// TIA Portal V18 export
DATA_BLOCK "L1_gen"   // DB3
{ S7_Optimized_Access := 'TRUE' }
VERSION : 0.1
// stored: AutoNumber true, DBAccessibleFromOPCUA true, DBAccessibleFromWebserver true, IsOnlyStoredInLoadMemory false, IsRetainMemResEnabled false, IsWriteProtectedInAS false, MemoryReserve 100
   VAR RETAIN
      linea { S7_SetPoint := 'True'} : "LGasp_typeHMI_linea";
   END_VAR
BEGIN
   linea.NUMZONE := 5;
   linea.NUMDS := 50;
   linea.NUMSTAZIONI := 20;
   linea.NUMSAFETYDEVICE := 15;
   linea.NUMATTUATORI := 15;
   linea.NUMPUNZONATEARTICOLO := 100;
   linea.NUMRIGHEPRODUZIONE := 10;
   linea.NUMRIGHELISTATAGLI := 50;
   linea.NUMASSIAA := 3;
   linea.man := FALSE;
   linea.auto := FALSE;
   linea.semiauto := FALSE;
   linea.MARCIAstop := FALSE;
   linea.allarmi := TRUE;
   linea.warning := TRUE;
   linea.nome_linea := WSTRING#'210100008';
   linea.zona[1].abilitata := TRUE;
   linea.zona[2].abilitata := FALSE;
   linea.zona[3..4].abilitata := TRUE;
   linea.zona[5].abilitata := FALSE;
   linea.zona[1].nome := WSTRING#'Z1';
   linea.zona[2].nome := WSTRING#'Z2';
   linea.zona[3].nome := WSTRING#'Z3';
   linea.zona[4].nome := WSTRING#'Z4';
   linea.zona[5].nome := WSTRING#'Z5';
   linea.zona[1..5].AUTOman := FALSE;
   linea.zona[1..5].MARCIAstop := FALSE;
   linea.zona[1].allarmi := TRUE;
   linea.zona[2].allarmi := FALSE;
   linea.zona[3].allarmi := TRUE;
   linea.zona[4..5].allarmi := FALSE;
   linea.zona[1..5].warning := FALSE;
   linea.zona[1..5].fungointervenuto := FALSE;
   linea.zona[1..5].cancellointervenuto := FALSE;
   linea.zona[1].barrieraintervenuta := TRUE;
   linea.zona[2..5].barrieraintervenuta := FALSE;
   linea.zona[1].safetydevice[1..3].tipo := 1;
   linea.zona[1].safetydevice[4].tipo := 3;
   linea.zona[1].safetydevice[5].tipo := 5;
   linea.zona[1].safetydevice[6..15].tipo := 0;
   linea.zona[2].safetydevice[1..15].tipo := 0;
   linea.zona[3].safetydevice[1..3].tipo := 1;
   linea.zona[3].safetydevice[4..5].tipo := 5;
   linea.zona[3].safetydevice[6..9].tipo := 1;
   linea.zona[3].safetydevice[10..12].tipo := 5;
   linea.zona[3].safetydevice[13..15].tipo := 0;
   linea.zona[4].safetydevice[1..2].tipo := 1;
   linea.zona[4].safetydevice[3..5].tipo := 6;
   linea.zona[4].safetydevice[6..15].tipo := 0;
   linea.zona[5].safetydevice[1..15].tipo := 0;
   linea.zona[1].safetydevice[1].conn := WSTRING#'XC100';
   linea.zona[1].safetydevice[2].conn := WSTRING#'XC101';
   linea.zona[1].safetydevice[3].conn := WSTRING#'XC105';
   linea.zona[1].safetydevice[4].conn := WSTRING#'XC142';
   linea.zona[1].safetydevice[5].conn := WSTRING#'XC701';
   linea.zona[1].safetydevice[6..15].conn := WSTRING#'';
   linea.zona[2].safetydevice[1..15].conn := WSTRING#'';
   linea.zona[3].safetydevice[1].conn := WSTRING#'XC141';
   linea.zona[3].safetydevice[2].conn := WSTRING#'XC162';
   linea.zona[3].safetydevice[3].conn := WSTRING#'XC803';
   linea.zona[3].safetydevice[4].conn := WSTRING#'XC702';
   linea.zona[3].safetydevice[5].conn := WSTRING#'XC703';
   linea.zona[3].safetydevice[6].conn := WSTRING#'QE1';
   linea.zona[3].safetydevice[7].conn := WSTRING#'QE2';
   linea.zona[3].safetydevice[8].conn := WSTRING#'XC305';
   linea.zona[3].safetydevice[9].conn := WSTRING#'XC50';
   linea.zona[3].safetydevice[10].conn := WSTRING#'XC704';
   linea.zona[3].safetydevice[11].conn := WSTRING#'XC705';
   linea.zona[3].safetydevice[12].conn := WSTRING#'XC706';
   linea.zona[3].safetydevice[13..15].conn := WSTRING#'';
   linea.zona[4].safetydevice[1].conn := WSTRING#'XC400';
   linea.zona[4].safetydevice[2].conn := WSTRING#'XC406';
   linea.zona[4].safetydevice[3].conn := WSTRING#'XC707';
   linea.zona[4].safetydevice[4].conn := WSTRING#'XC708';
   linea.zona[4].safetydevice[5..15].conn := WSTRING#'';
   linea.zona[5].safetydevice[1..15].conn := WSTRING#'';
   linea.zona[1].safetydevice[1..3].intervenuto := FALSE;
   linea.zona[1].safetydevice[4].intervenuto := TRUE;
   linea.zona[1].safetydevice[5..15].intervenuto := FALSE;
   linea.zona[2].safetydevice[1].intervenuto := FALSE;
   linea.zona[2].safetydevice[2].intervenuto := TRUE;
   linea.zona[2].safetydevice[3..15].intervenuto := FALSE;
   linea.zona[3].safetydevice[1..15].intervenuto := FALSE;
   linea.zona[4].safetydevice[1..4].intervenuto := FALSE;
   linea.zona[4].safetydevice[5].intervenuto := TRUE;
   linea.zona[4].safetydevice[6..15].intervenuto := FALSE;
   linea.zona[5].safetydevice[1..2].intervenuto := FALSE;
   linea.zona[5].safetydevice[3..4].intervenuto := TRUE;
   linea.zona[5].safetydevice[5..15].intervenuto := FALSE;
   linea.zona[1].safetydevice[1..5].ninterventi := 2;
   linea.zona[1].safetydevice[6..15].ninterventi := 0;
   linea.zona[2].safetydevice[1].ninterventi := 4;
   linea.zona[2].safetydevice[2].ninterventi := 5;
   linea.zona[2].safetydevice[3].ninterventi := 4;
   linea.zona[2].safetydevice[4..7].ninterventi := 5;
   linea.zona[2].safetydevice[8..15].ninterventi := 0;
   linea.zona[3].safetydevice[1..8].ninterventi := 2;
   linea.zona[3].safetydevice[9].ninterventi := 3;
   linea.zona[3].safetydevice[10..12].ninterventi := 2;
   linea.zona[3].safetydevice[13..15].ninterventi := 0;
   linea.zona[4].safetydevice[1].ninterventi := 3;
   linea.zona[4].safetydevice[2..4].ninterventi := 2;
   linea.zona[4].safetydevice[5].ninterventi := 9;
   linea.zona[4].safetydevice[6..15].ninterventi := 0;
   linea.zona[5].safetydevice[1..2].ninterventi := 4;
   linea.zona[5].safetydevice[3].ninterventi := 7;
   linea.zona[5].safetydevice[4].ninterventi := 9;
   linea.zona[5].safetydevice[5..15].ninterventi := 0;
   linea.zona[1].safetydevice[1..15].dadefinire1 := 0;
   linea.zona[2].safetydevice[1..15].dadefinire1 := 0;
   linea.zona[3].safetydevice[1..15].dadefinire1 := 0;
   linea.zona[4].safetydevice[1..15].dadefinire1 := 0;
   linea.zona[5].safetydevice[1..15].dadefinire1 := 0;
   linea.zona[1].safetydevice[1..15].dadefinire2 := 0;
   linea.zona[2].safetydevice[1..15].dadefinire2 := 0;
   linea.zona[3].safetydevice[1..15].dadefinire2 := 0;
   linea.zona[4].safetydevice[1..15].dadefinire2 := 0;
   linea.zona[5].safetydevice[1..15].dadefinire2 := 0;
   linea.zona[1].safetydevice[1..15].dadefinire3 := 0;
   linea.zona[2].safetydevice[1..15].dadefinire3 := 0;
   linea.zona[3].safetydevice[1..15].dadefinire3 := 0;
   linea.zona[4].safetydevice[1..15].dadefinire3 := 0;
   linea.zona[5].safetydevice[1..15].dadefinire3 := 0;
   // linea.stz[1] : QUADRO
   // linea.stz[2] : PROFINET
   // linea.stz[3] : GENERALE
   // linea.stz[4] : ASPO+CULLA
   // linea.stz[5] : RADDRIZZATRICE
   // linea.stz[6] : GIUNZIONE
   // linea.stz[7] : ALIM+PUNZ
   // linea.stz[8] : PROFILA
   // linea.stz[9] : TAGLIO
   // linea.stz[10] : SCARICO
   linea.stz[1..10].abilitata := TRUE;
   linea.stz[11..20].abilitata := FALSE;
   linea.stz[1..2].invisibile := TRUE;
   linea.stz[3..5].invisibile := FALSE;
   linea.stz[6..7].invisibile := TRUE;
   linea.stz[8..9].invisibile := FALSE;
   linea.stz[10..20].invisibile := TRUE;
   linea.stz[1..3].zona := 3;
   linea.stz[4].zona := 1;
   linea.stz[5..7].zona := 2;
   linea.stz[8].zona := 3;
   linea.stz[9].zona := 4;
   linea.stz[10..20].zona := 5;
   linea.stz[1].nome := WSTRING#'STZ QUADRO';
   linea.stz[2].nome := WSTRING#'STZ PROFINET';
   linea.stz[3].nome := WSTRING#'STZ GENERALE';
   linea.stz[4].nome := WSTRING#'STZ ASPO+CULLA';
   linea.stz[5].nome := WSTRING#'STZ RADDRIZZATRICE';
   linea.stz[6].nome := WSTRING#'STZ GIUNZIONE';
   linea.stz[7].nome := WSTRING#'STZ ALIM+PUNZ';
   linea.stz[8].nome := WSTRING#'STZ PROFILA';
   linea.stz[9].nome := WSTRING#'STZ TAGLIO';
   linea.stz[10].nome := WSTRING#'STZ SCARICO';
   linea.stz[11..20].nome := WSTRING#'';
   linea.stz[1].nometrad := WSTRING#'QUADRO';
   linea.stz[2].nometrad := WSTRING#'PROFINET';
   linea.stz[3].nometrad := WSTRING#'GENERALE';
   linea.stz[4].nometrad := WSTRING#'ASPO';
   linea.stz[5].nometrad := WSTRING#'RADDRIZZATRICE';
   linea.stz[6].nometrad := WSTRING#'GIUNZIONE';
   linea.stz[7].nometrad := WSTRING#'ALIM + PUNZ';
   linea.stz[8].nometrad := WSTRING#'PROFILA';
   linea.stz[9].nometrad := WSTRING#'TAGLIO';
   linea.stz[10].nometrad := WSTRING#'SCARICO';
   linea.stz[11].nometrad := WSTRING#'AGGRAFFATURA';
   linea.stz[12..19].nometrad := WSTRING#'DISPONIBILE';
   linea.stz[20].nometrad := WSTRING#'';
   linea.stz[1..20].AUTOman := FALSE;
   linea.stz[1..20].MARCIAstop := FALSE;
   linea.stz[1..2].allarmi := FALSE;
   linea.stz[3..4].allarmi := TRUE;
   linea.stz[5..7].allarmi := FALSE;
   linea.stz[8].allarmi := TRUE;
   linea.stz[9..20].allarmi := FALSE;
   linea.stz[1..3].warning := FALSE;
   linea.stz[4].warning := TRUE;
   linea.stz[5..20].warning := FALSE;
   // linea.stz[4].ds[1] : L1-ASPO- DIAMETRO COIL-DISTANZA LASER CENTRO ASPO [mm]
   // linea.stz[4].ds[2] : L1-ASPO- ANSA XC142A-1-SOGLIA BASSA [mm]
   // linea.stz[4].ds[3] : L1-ASPO- ANSA XC142A-1-SOGLIA ALTA [mm]
   // linea.stz[4].ds[5] : L1-ASPO-FRENATURA-COPPIA MAX [%]
   // linea.stz[4].ds[6] : L1-ASPO-FRENATURA-VELOCITA' AUTOMATICA [%]
   // linea.stz[4].ds[8] : L1-ASPO-M101 MADRINO -VELOCITA' MANUALE [%]
   // linea.stz[4].ds[15] : L1-ASPO-M101 MADRINO -INTERVALLO PER ESPANSIONE AUTOMATICA [min]
   // linea.stz[4].ds[16] : L1-ASPO-M101 MADRINO -DURATA ESPANSIONE AUTOMATICA [sec]
   // linea.stz[5].ds[1] : L1-RADDRIZZATRICE-ANSA-VELOCITA' BASSA [%]
   // linea.stz[5].ds[2] : L1-RADDRIZZATRICE-ANSA-VELOCITA' MEDIA [%]
   // linea.stz[5].ds[3] : L1-RADDRIZZATRICE-ANSA-VELOCITA' ALTA [%]
   // linea.stz[5].ds[4] : L1-RADDRIZZATRICE-ANSA-SOGLIA BASSA [mm]
   // linea.stz[5].ds[5] : L1-RADDRIZZATRICE-ANSA-SOGLIA INTEMEDIA BASSA [mm]
   // linea.stz[5].ds[6] : L1-RADDRIZZATRICE-ANSA-SOGLIA INTEMEDIA ALTA [mm]
   // linea.stz[5].ds[7] : L1-RADDRIZZATRICE-ANSA-SOGLIA ALTA [mm]
   // linea.stz[5].ds[8] : L1-RADDRIZZATRICE-M141-VELOCITA' MANUALE [%]
   // linea.stz[7].ds[1] : L1-ALIM + PUNZ-M201-ALIMENTATORE A RULLI-VELOCITA' MANUALE [%]
   // linea.stz[7].ds[2] : L1-ALIM + PUNZ-M201-ALIMENTATORE A RULLI-VELOCITA QUOTA FINE PRODUZIONE [%]
   // linea.stz[7].ds[3] : L1-ALIM + PUNZ-M201-ALIMENTATORE A RULLI-DISTANZA LAMA-GIUNZIONE CON PUNTO DI SALDATURA [mm]
   // linea.stz[7].ds[4] : L1-ALIM + PUNZ-M201-ALIMENTATORE A RULLI-QUOTA ALIMENTATORE A FINE PRODUZIONE [mm]
   // linea.stz[7].ds[5] : L1-ALIM + PUNZ-ANSA-SOGLIA BASSA [mm]
   // linea.stz[7].ds[6] : L1-ALIM + PUNZ-ANSA-SOGLIA INTEMEDIA BASSA [mm]
   // linea.stz[7].ds[7] : L1-ALIM + PUNZ-ANSA-SOGLIA INTEMEDIA ALTA [mm]
   // linea.stz[7].ds[8] : L1-ALIM + PUNZ-ANSA-SOGLIA ALTA [mm]
   // linea.stz[7].ds[9] : L1-ALIM + PUNZ-PRESSA-VELOCITA MANUALE-SEMIAUTO [%]
   // linea.stz[7].ds[10] : L1-ALIM + PUNZ-PRESSA-OFFSET ENCODER ASSOLUTO
   // linea.stz[7].ds[11] : L1-ALIM + PUNZ-PRESSA-ANGOLO INIZIO PMS [°]
   // linea.stz[7].ds[12] : L1-ALIM + PUNZ-PRESSA-ANGOLO FINE PMS [°]
   // linea.stz[7].ds[13] : L1-ALIM + PUNZ-PRESSA-ANGOLO INIZIO PMI [°]
   // linea.stz[7].ds[14] : L1-ALIM + PUNZ-PRESSA-ANGOLO FINE PMI [°]
   // linea.stz[7].ds[15] : L1-ALIM + PUNZ-PRESSA-ANGOLO INIZIO AREA DI LAVORO [°]
   // linea.stz[7].ds[16] : L1-ALIM + PUNZ-PRESSA-ANGOLO FINE AREA DI LAVORO [°]
   // linea.stz[7].ds[17] : L1-ALIM + PUNZ-PRESSA-NUMERO COLPI IN SEMI AUTOMATICO
   // linea.stz[7].ds[18] : L1-ALIM + PUNZ-DROPSA-NUMERO COLPI PER LUBRIFICAZIONE
   // linea.stz[7].ds[19] : L1-ALIM + PUNZ-DROPSA-DURATA LUBRIFICAZIONE [sec]
   // linea.stz[8].ds[1] : L1-PROFILA-M301 PROFILA-VELOCITA' MANUALE [%]
   // linea.stz[8].ds[2] : L1-PROFILA-M301 PROFILA-VELOCITA SVUOTAMENTO [%]
   // linea.stz[8].ds[4] : L1-PROFILA-M365 ESTRATTORE-VELOCITA' MANUALE [%]
   // linea.stz[8].ds[8] : L1-PROFILA-SALDATRICE-POTENZA SALDATURA [%]
   // linea.stz[8].ds[11] : L1-PROFILA-QUOTA ATTIVAZIONE LUBRIFICAZIONE [mm]
   // linea.stz[8].ds[12] : L1-PROFILA-DURATA LUBRIFICAZIONE [sec]
   // linea.stz[9].ds[2] : L1-TAGLIO-DURATA LUBRIFICAZIONE [sec]
   // linea.stz[9].ds[3] : L1-TAGLIO-NUMERO COLPI PER LUBRIFICAZIONE
   // linea.stz[9].ds[4] : L1-TAGLIO-M404 SALITA DISCESA DISCO TAGLIO-VELOCITA' MANUALE [%]
   // linea.stz[9].ds[6] : L1-TAGLIO-M405 ROTAZIONE DISCO TAGLIO-VELOCITA' MANUALE [%]
   // linea.stz[9].ds[7] : L1-TAGLIO-M405 ROTAZIONE DISCO TAGLIO-VELOCITA' SPESSORE 0.5-0.6
   // linea.stz[9].ds[8] : L1-TAGLIO-M405 ROTAZIONE DISCO TAGLIO-VELOCITA' SPESSORE 0.8-1.0
   // linea.stz[9].ds[9] : L1-TAGLIO-M405 ROTAZIONE DISCO TAGLIO-VELOCITA' SPESSORE 1.2-1.5
   // linea.stz[9].ds[10] : L1-TAGLIO-M404 SALITA DISCESA DISCO TAGLIO-POSIZIONE PUNTO MORTO SUP [mm]
   // linea.stz[9].ds[11] : L1-TAGLIO-M404 SALITA DISCESA DISCO TAGLIO-POSIZIONE PUNTO MORTO INF [mm]
   // linea.stz[9].ds[12] : L1-TAGLIO-M404 SALITA DISCESA DISCO TAGLIO-POSIZIONE CAMBIO LAMA [mm]
   // linea.stz[9].ds[13] : L1-TAGLIO-M404 SALITA DISCESA DISCO TAGLIO-VELOCITA' SPESSORE 0.5-0.6
   // linea.stz[9].ds[14] : L1-TAGLIO-M404 SALITA DISCESA DISCO TAGLIO-VELOCITA' SPESSORE 0.8-1.0
   // linea.stz[9].ds[15] : L1-TAGLIO-M404 SALITA DISCESA DISCO TAGLIO-VELOCITA' SPESSORE 1.2-1.5
   // linea.stz[9].ds[16] : L1-TAGLIO-M404 SALITA DISCESA DISCO TAGLIO-VELOCITA' SALITA
   // linea.stz[9].ds[17] : L1-TAGLIO-M401 CARRO TAGLIO AL VOLO-DISTANZA LASER LAMA DI TAGLIO[mm]
   // linea.stz[9].ds[19] : L1-TAGLIO-M408 TAPPETO EVACUAZIONE-VELOCITA INTERMEDIA [%]
   // linea.stz[9].ds[20] : L1-TAGLIO-M408 TAPPETO EVACUAZIONE-VELOCITA' ALTA [%]
   // linea.stz[9].ds[21] : L1-TAGLIO-M408 TAPPETO EVACUAZIONE-VELOCITA' MANUALE [%]
   linea.stz[1].ds[1..50].val := 0.0;
   linea.stz[2].ds[1..50].val := 0.0;
   linea.stz[3].ds[1..50].val := 0.0;
   linea.stz[4].ds[1].val := 2090.0;
   linea.stz[4].ds[2..4].val := 0.0;
   linea.stz[4].ds[5].val := 10.0;
   linea.stz[4].ds[6].val := 1.0;
   linea.stz[4].ds[7].val := 0.0;
   linea.stz[4].ds[8..9].val := 10.0;
   linea.stz[4].ds[10..12].val := 25.0;
   linea.stz[4].ds[13..14].val := 0.0;
   linea.stz[4].ds[15].val := 5.0;
   linea.stz[4].ds[16].val := 60.0;
   linea.stz[4].ds[17].val := 0.0;
   linea.stz[4].ds[18].val := 5.0;
   linea.stz[4].ds[19].val := 60.0;
   linea.stz[4].ds[20..50].val := 0.0;
   linea.stz[5].ds[1].val := 5.0;
   linea.stz[5].ds[2].val := 50.0;
   linea.stz[5].ds[3].val := 80.0;
   linea.stz[5].ds[4].val := 2300.0;
   linea.stz[5].ds[5].val := 2200.0;
   linea.stz[5].ds[6].val := 2000.0;
   linea.stz[5].ds[7].val := 1700.0;
   linea.stz[5].ds[8].val := 80.0;
   linea.stz[5].ds[9..50].val := 0.0;
   linea.stz[6].ds[1..50].val := 0.0;
   linea.stz[7].ds[1].val := 20.0;
   linea.stz[7].ds[2..4].val := 0.0;
   linea.stz[7].ds[5].val := 2300.0;
   linea.stz[7].ds[6].val := 2200.0;
   linea.stz[7].ds[7].val := 2000.0;
   linea.stz[7].ds[8].val := 1700.0;
   linea.stz[7].ds[9].val := 60.0;
   linea.stz[7].ds[10].val := -214.0;
   linea.stz[7].ds[11].val := 340.0;
   linea.stz[7].ds[12].val := 20.0;
   linea.stz[7].ds[13].val := 160.0;
   linea.stz[7].ds[14].val := 200.0;
   linea.stz[7].ds[15].val := 130.0;
   linea.stz[7].ds[16].val := 230.0;
   linea.stz[7].ds[17].val := 60.0;
   linea.stz[7].ds[18..50].val := 0.0;
   linea.stz[8].ds[1].val := 15.0;
   linea.stz[8].ds[2].val := 10.0;
   linea.stz[8].ds[3..4].val := 0.0;
   linea.stz[8].ds[5].val := 10000.0;
   linea.stz[8].ds[6].val := 30.0;
   linea.stz[8].ds[7].val := 0.0;
   linea.stz[8].ds[8].val := 90.0;
   linea.stz[8].ds[9..10].val := 0.0;
   linea.stz[8].ds[11].val := 60.0;
   linea.stz[8].ds[12..13].val := 1.0;
   linea.stz[8].ds[14..50].val := 0.0;
   linea.stz[9].ds[1..50].val := 0.0;
   linea.stz[10].ds[1..50].val := 0.0;
   linea.stz[11].ds[1..50].val := 0.0;
   linea.stz[12].ds[1..50].val := 0.0;
   linea.stz[13].ds[1..50].val := 0.0;
   linea.stz[14].ds[1..50].val := 0.0;
   linea.stz[15].ds[1..50].val := 0.0;
   linea.stz[16].ds[1..50].val := 0.0;
   linea.stz[17].ds[1..50].val := 0.0;
   linea.stz[18].ds[1..50].val := 0.0;
   linea.stz[19].ds[1..50].val := 0.0;
   linea.stz[20].ds[1..50].val := 0.0;
   linea.stz[1].ds[1..50].ll := 0.0;
   linea.stz[2].ds[1..50].ll := 0.0;
   linea.stz[3].ds[1..50].ll := 0.0;
   linea.stz[4].ds[1..4].ll := 0.0;
   linea.stz[4].ds[5..6].ll := 1.0;
   linea.stz[4].ds[7..9].ll := 0.0;
   linea.stz[4].ds[10..12].ll := 1.0;
   linea.stz[4].ds[13..50].ll := 0.0;
   linea.stz[5].ds[1..50].ll := 0.0;
   linea.stz[6].ds[1..50].ll := 0.0;
   linea.stz[7].ds[1..9].ll := 0.0;
   linea.stz[7].ds[10].ll := -360.0;
   linea.stz[7].ds[11..16].ll := 0.0;
   linea.stz[7].ds[17].ll := 40.0;
   linea.stz[7].ds[18..50].ll := 0.0;
   linea.stz[8].ds[1..2].ll := 1.0;
   linea.stz[8].ds[3..5].ll := 0.0;
   linea.stz[8].ds[6].ll := 1.0;
   linea.stz[8].ds[7].ll := 0.0;
   linea.stz[8].ds[8].ll := 1.0;
   linea.stz[8].ds[9..12].ll := 0.0;
   linea.stz[8].ds[13].ll := 0.9;
   linea.stz[8].ds[14..50].ll := 0.0;
   linea.stz[9].ds[1..50].ll := 0.0;
   linea.stz[10].ds[1..50].ll := 0.0;
   linea.stz[11].ds[1..50].ll := 0.0;
   linea.stz[12].ds[1..50].ll := 0.0;
   linea.stz[13].ds[1..50].ll := 0.0;
   linea.stz[14].ds[1..50].ll := 0.0;
   linea.stz[15].ds[1..50].ll := 0.0;
   linea.stz[16].ds[1..50].ll := 0.0;
   linea.stz[17].ds[1..50].ll := 0.0;
   linea.stz[18].ds[1..50].ll := 0.0;
   linea.stz[19].ds[1..50].ll := 0.0;
   linea.stz[20].ds[1..50].ll := 0.0;
   linea.stz[1].ds[1..50].hl := 0.0;
   linea.stz[2].ds[1..50].hl := 0.0;
   linea.stz[3].ds[1..50].hl := 0.0;
   linea.stz[4].ds[1].hl := 3000.0;
   linea.stz[4].ds[2..4].hl := 0.0;
   linea.stz[4].ds[5..6].hl := 100.0;
   linea.stz[4].ds[7].hl := 0.0;
   linea.stz[4].ds[8..12].hl := 100.0;
   linea.stz[4].ds[13..14].hl := 0.0;
   linea.stz[4].ds[15].hl := 60.0;
   linea.stz[4].ds[16].hl := 200.0;
   linea.stz[4].ds[17].hl := 0.0;
   linea.stz[4].ds[18].hl := 60.0;
   linea.stz[4].ds[19].hl := 200.0;
   linea.stz[4].ds[20..50].hl := 0.0;
   linea.stz[5].ds[1..3].hl := 100.0;
   linea.stz[5].ds[4..7].hl := 2400.0;
   linea.stz[5].ds[8].hl := 100.0;
   linea.stz[5].ds[9..50].hl := 0.0;
   linea.stz[6].ds[1..50].hl := 0.0;
   linea.stz[7].ds[1].hl := 100.0;
   linea.stz[7].ds[2..4].hl := 0.0;
   linea.stz[7].ds[5..8].hl := 2400.0;
   linea.stz[7].ds[9].hl := 100.0;
   linea.stz[7].ds[10..16].hl := 360.0;
   linea.stz[7].ds[17].hl := 100.0;
   linea.stz[7].ds[18..50].hl := 0.0;
   linea.stz[8].ds[1..2].hl := 100.0;
   linea.stz[8].ds[3..4].hl := 0.0;
   linea.stz[8].ds[5].hl := 20000.0;
   linea.stz[8].ds[6].hl := 100.0;
   linea.stz[8].ds[7].hl := 0.0;
   linea.stz[8].ds[8].hl := 100.0;
   linea.stz[8].ds[9..10].hl := 0.0;
   linea.stz[8].ds[11].hl := 120.0;
   linea.stz[8].ds[12].hl := 60.0;
   linea.stz[8].ds[13].hl := 1.1;
   linea.stz[8].ds[14..50].hl := 0.0;
   linea.stz[9].ds[1..22].hl := 0.0;
   linea.stz[9].ds[23].hl := 2000.0;
   linea.stz[9].ds[24..50].hl := 0.0;
   linea.stz[10].ds[1..50].hl := 0.0;
   linea.stz[11].ds[1..50].hl := 0.0;
   linea.stz[12].ds[1..50].hl := 0.0;
   linea.stz[13].ds[1..50].hl := 0.0;
   linea.stz[14].ds[1..50].hl := 0.0;
   linea.stz[15].ds[1..50].hl := 0.0;
   linea.stz[16].ds[1..50].hl := 0.0;
   linea.stz[17].ds[1..50].hl := 0.0;
   linea.stz[18].ds[1..50].hl := 0.0;
   linea.stz[19].ds[1..50].hl := 0.0;
   linea.stz[20].ds[1..50].hl := 0.0;
   linea.stz[1].all[1] := FALSE;   // L1-QUADRO[1]- 24-L4+ EMERGENZA GENERALE
   linea.stz[1].all[2] := FALSE;   // L1-QUADRO[2]-
   linea.stz[1].all[3] := FALSE;   // L1-QUADRO[3]-D6-QF1-PROTEZIONE INTERVENUTA PRIMARIO TRASFORMATORE 400:230V
   linea.stz[1].all[4] := FALSE;   // L1-QUADRO[4]-D6-QF2-PROTEZIONE INTERVENUTA SECONDARIO TRASFORMATORE 400:230V
   linea.stz[1].all[5] := FALSE;
   linea.stz[1].all[6] := FALSE;   // L1-QUADRO[6]-D8-FU1 24-L1+-PROTEZIONE ELETTRONICA INTERVENUTA ALIMENTAZIONE Q.E.
   linea.stz[1].all[7] := FALSE;   // L1-QUADRO[7]-D8 FU1 24-L3+-PROTEZIONE ELETTRONICA INTERVENUTA ALIMENTAZIONE PULSANTIERE
   linea.stz[1].all[8] := FALSE;   // L1-QUADRO[8]-D8 FU1 24-L3+S-PROTEZIONE ELETTRONICA INTERVENUTA ALIMENTAZIONE SICUREZZE
   linea.stz[1].all[9] := FALSE;   // L1-QUADRO[9]-D8 FU1 24-L3+1-PROTEZIONE ELETTRONICA INTERVENUTA ALIMENTAZIONE B.M.1 (MANDRINI ASPO)
   linea.stz[1].all[10] := FALSE;   // L1-QUADRO[10]-D8 FU1 24-L3+2-PROTEZIONE ELETTRONICA INTERVENUTA ALIMENTAZIONE B.M. 2 (TIN + RADDRIZZATRICE- + CENTRALE PROFILA)
   linea.stz[1].all[11] := FALSE;   // L1-QUADRO[11]-D8 FU1 24-L3+3-PROTEZIONE ELETTRONICA INTERVENUTA ALIMENTAZIONE B.M. 3 (VASCA LIQUIDO)
   linea.stz[1].all[12] := FALSE;   // L1-QUADRO[12]-D8 FU1 24-L10+-PROTEZIONE ELETTRONICA INTERVENUTA ALIMENTAZIONE PC
   linea.stz[1].all[13] := FALSE;   // L1-QUADRO[13]-D8 FU1 24-L11+ PROTEZIONE ELETTRONICA INTERVENUTA ALIMENTAZIONE NODI IN Q.E.
   linea.stz[1].all[14] := FALSE;   // L1-QUADRO[14]-D9 FU1 24-L13+ -PROTEZIONE ELETTRONICA INTERVENUTA ALIMENTAZIONE LOGICA AZIONAMENTI
   linea.stz[1].all[15] := FALSE;   // L1-QUADRO[15]-D9 FU1 24-L131+ -PROTEZIONE ELETTRONICA INTERVENUTA ALIMENTAZIONE LOGICA ALIMENTATORE 45KW
   linea.stz[1].all[16] := FALSE;   // L1-QUADRO[16]-D9 FU124-L3+4 PROTEZIONE ELETTRONICA INTERVENUTA ALIMENTAZIONE B.M. 4 (TAGLIO + CENTRALE IDRAULICA)
   linea.stz[1].all[17] := FALSE;   // L1-QUADRO[17]-D17 FU1 OUT 4 (PREDISPOSTO)
   linea.stz[1].all[18] := FALSE;   // L1-QUADRO[18]-D16 FU1 24-L4+ PROTEZIONE ELETTRONICA INTERVENUTA - EMERGENZA GENERALE
   linea.stz[1].all[19] := FALSE;   // L1-QUADRO[19]-D16 FU1 24-L41+ PROTEZIONE ELETTRONICA INTERVENUTA - EMERGENZA ISTANTANEA ZONA 1 (SVOLGITURA)
   linea.stz[1].all[20] := FALSE;   // L1-QUADRO[20]-D16 FU1 24-L42+ PROTEZIONE ELETTRONICA INTERVENUTA - EMERGENZA ISTANTANEA ZONA 2 (GIUNZIONE)
   linea.stz[1].all[21] := FALSE;   // L1-QUADRO[21]-D16 FU1 24-L44+ PROTEZIONE ELETTRONICA INTERVENUTA - EMERGENZA ISTANTANEA ZONA 4 TAGLIO)
   linea.stz[1].all[22] := FALSE;   // L1-QUADRO[22]-D16 FU1 24-L43+ PROTEZIONE ELETTRONICA INTERVENUTA - EMERGENZA ISTANTANEA ZONA 3 PROFILA)
   linea.stz[1].all[23] := FALSE;   // L1-QUADRO[23]-D16 FU1 24-L411+ PROTEZIONE ELETTRONICA INTERVENUTA - EMERGENZA ISTANTANEA ZONA 1 MANDRINO 1)
   linea.stz[1].all[24] := FALSE;   // L1-QUADRO[24]-D16 FU1 24-L412+ PROTEZIONE ELETTRONICA INTERVENUTA - EMERGENZA ISTANTANEA ZONA 1 MANDRINO 2)
   linea.stz[1].all[25] := FALSE;   // L1-QUADRO[25]-D16 FU1 24-L4+3 PROTEZIONE ELETTRONICA INTERVENUTA - EMERGENZA ISTANTANEA
   linea.stz[1].all[26] := FALSE;   // L1-QUADRO[26]-D17 FU1 24-L4+1 PROTEZIONE ELETTRONICA INTERVENUTA - EMERGENZA ISTANTANEA
   linea.stz[1].all[27] := FALSE;   // L1-QUADRO[27]-D17 FU1 24-L4+2 PROTEZIONE ELETTRONICA INTERVENUTA - EMERGENZA ISTANTANEA
   linea.stz[1].all[28] := FALSE;   // L1-QUADRO[28]-D17 FU1 24-L43+1 PROTEZIONE ELETTRONICA INTERVENUTA - EMERGENZA ISTANTANEA
   linea.stz[1].all[29] := FALSE;   // L1-QUADRO[29]-D17 OUT 4 PREDISPOSTO
   linea.stz[1].all[30] := FALSE;   // L1-QUADRO[30]-D7-QF1 TERMICA ALIMENTATORE LINEA 24VDC INGRESSI
   linea.stz[1].all[31] := FALSE;   // L1-QUADRO[31]- D15-QF1 TERMICA ALIMENTATORE LINEA 24VDC USCITE
   linea.stz[1].all[32] := FALSE;   // L1-QUADRO[32]-D21-QF1 LINEA TERMICA PRESE QUADRO ELETTRICO
   linea.stz[1].all[33] := FALSE;   // L1-QUADRO[33]- D23-QF1 TERMICA VENTILAZIONE QUADRO
   linea.stz[1].all[34] := FALSE;   // L1-QUADRO[34]- D15-UV1 ANOMALIA ALIMENTATORE 1
   linea.stz[1].all[35] := FALSE;   // L1-QUADRO[35]- D15-UV2 ANOMALIA ALIMENTATORE 2
   linea.stz[1].all[36] := FALSE;   // L1-QUADRO[36]-
   linea.stz[1].all[37] := FALSE;   // L1-QUADRO[37]-
   linea.stz[1].all[38] := FALSE;   // L1-QUADRO[38]- G13-QF361 TERMICA MOTORE POMPA MANDATA LUBROREFRIGERAZIONE
   linea.stz[1].all[39] := FALSE;   // L1-QUADRO[39]- G14-QF368 TERMICA MOTORE POMPA SOMMERSA LUBROREFRIGERAZIONE
   linea.stz[1].all[40] := FALSE;   // L1-QUADRO[40]-
   linea.stz[1].all[41] := FALSE;   // L1-QUADRO[41]-
   linea.stz[1].all[42] := FALSE;   // L1-QUADRO[42]-
   linea.stz[1].all[43] := FALSE;   // L1-QUADRO[43]-
   linea.stz[1].all[44] := FALSE;   // L1-QUADRO[44]- M7-BT1- ALTA TEMPERATURA
   linea.stz[1].all[45] := FALSE;   // L1-QUADRO[45]-
   linea.stz[1].all[46] := FALSE;   // L1-QUADRO[46]-
   linea.stz[1].all[47] := FALSE;   // L1-QUADRO[47]-
   linea.stz[1].all[48] := FALSE;   // L1-QUADRO[48]-
   linea.stz[1].all[49] := FALSE;   // L1-QUADRO[49]-
   linea.stz[1].all[50] := FALSE;   // L1-QUADRO[50]-
   linea.stz[1].all[51] := FALSE;   // L1-QUADRO[51]-
   linea.stz[1].all[52] := FALSE;   // L1-QUADRO[52]
   linea.stz[1].all[53] := FALSE;   // L1-QUADRO[53]
   linea.stz[1].all[54] := FALSE;   // L1-QUADRO[54]-
   linea.stz[1].all[55..59] := FALSE;
   linea.stz[1].all[60] := FALSE;   // L1-QUADRO[60]-M9-M112-141DRV SOGLIA CARICO TERMICO RESISTENZA FRENATURA TORRETTA E RADDRIZZATORE
   linea.stz[1].all[61] := FALSE;   // L1-QUADRO[61]-M9-M102DRV SOGLIA CARICO TERMICO RESISTENZA FRENATURA ROTAZIONE MANDRINO 2
   linea.stz[1].all[62] := FALSE;   // L1-QUADRO[62]-M9-M101DRV SOGLIA CARICO TERMICO RESISTENZA FRENATURA ROTAZIONE MANDRINO 1
   linea.stz[1].all[63] := FALSE;   // L1-QUADRO[63]-M9-M401DRV SOGLIA CARICO TERMICO RESISTENZA FRENATURA TAGLIO ALVOLO
   linea.stz[1].all[64] := FALSE;   // L1-QUADRO[64]-M9-K30A1 ALTA TEMPERATURA ALIMENTATORE DRIVER 120KW
   linea.stz[1].all[65] := FALSE;   // L1-QUADRO[65]-M9-K30A1 ALIMENTATORE DRIVER BUS DC 120KW NON OK
   linea.stz[1].all[66] := FALSE;   // L1-QUADRO[66]-M9-K30A1 ALIMENTATORE DRIVER 120KW NON OK
   linea.stz[1].all[67] := FALSE;   // L1-QUADRO[67]-M10-M301DRV SOGLIA CARICO TERMICO RESISTENZA FRENATURA PROFILA MOTORE 1
   linea.stz[1].all[68] := FALSE;   // L1-QUADRO[68]-M10-M302DRV SOGLIA CARICO TERMICO RESISTENZA FRENATURA PROFILA MOTORE 2
   linea.stz[1].all[69] := FALSE;   // L1-QUADRO[69]-M10-M303DRV SOGLIA CARICO TERMICO RESISTENZA FRENATURA PROFILA MOTORE 3
   linea.stz[1].all[70] := FALSE;   // L1-QUADRO[70]- DIFFERENZIALE INTERVENUTO
   linea.stz[1].all[71] := FALSE;   // L1-QUADRO[71]-
   linea.stz[1].all[72] := FALSE;   // L1-QUADRO[72]-
   linea.stz[1].all[73] := FALSE;   // L1-QUADRO[73]-
   linea.stz[1].all[74] := FALSE;   // L1-QUADRO[74]-
   linea.stz[1].all[75] := FALSE;   // L1-QUADRO[75]-
   linea.stz[1].all[76] := FALSE;   // L1-QUADRO[76]-
   linea.stz[1].all[77] := FALSE;   // L1-QUADRO[77]-
   linea.stz[1].all[78] := FALSE;   // L1-QUADRO[78]-
   linea.stz[1].all[79] := FALSE;   // L1-QUADRO[79]-
   linea.stz[1].all[80] := FALSE;   // L1-QUADRO[80]-
   linea.stz[1].all[81..192] := FALSE;
   linea.stz[2].all[1] := FALSE;   // L1-PROFINET[1]
   linea.stz[2].all[2] := FALSE;   // L1-PROFINET[2]
   linea.stz[2].all[3] := FALSE;   // L1-PROFINET[3]
   linea.stz[2].all[4] := FALSE;   // L1-PROFINET[4]
   linea.stz[2].all[5] := FALSE;   // L1-PROFINET[5]
   linea.stz[2].all[6] := FALSE;   // L1-PROFINET[6]
   linea.stz[2].all[7] := FALSE;   // L1-PROFINET[7]
   linea.stz[2].all[8] := FALSE;   // L1-PROFINET[8]
   linea.stz[2].all[9] := FALSE;   // L1-PROFINET[9]
   linea.stz[2].all[10] := FALSE;   // L1-PROFINET[10]
   linea.stz[2].all[11] := FALSE;   // L1-PROFINET[11]
   linea.stz[2].all[12] := FALSE;   // L1-PROFINET[12]-ERRORE COMUNICAZIONE
   linea.stz[2].all[13] := FALSE;   // L1-PROFINET[13]
   linea.stz[2].all[14] := FALSE;   // L1-PROFINET[14]
   linea.stz[2].all[15] := FALSE;   // L1-PROFINET[15]
   linea.stz[2].all[16] := FALSE;   // L1-PROFINET[16]
   linea.stz[2].all[17] := FALSE;   // L1-PROFINET[17]
   linea.stz[2].all[18] := FALSE;   // L1-PROFINET[18]
   linea.stz[2].all[19] := FALSE;   // L1-PROFINET[19]
   linea.stz[2].all[20] := FALSE;   // L1-PROFINET[20]-ERRORE COMUNICAZIONE
   linea.stz[2].all[21] := FALSE;   // L1-PROFINET[21]-ERRORE COMUNICAZIONE
   linea.stz[2].all[22] := FALSE;   // L1-PROFINET[22]-ERRORE COMUNICAZIONE
   linea.stz[2].all[23] := FALSE;   // L1-PROFINET[23]-ERRORE COMUNICAZIONE
   linea.stz[2].all[24] := FALSE;   // L1-PROFINET[24]-ERRORE COMUNICAZIONE
   linea.stz[2].all[25] := FALSE;   // L1-PROFINET[25]
   linea.stz[2].all[26] := FALSE;   // L1-PROFINET[26]-ERRORE COMUNICAZIONE
   linea.stz[2].all[27] := FALSE;   // L1-PROFINET[27]
   linea.stz[2].all[28] := FALSE;   // L1-PROFINET[28]
   linea.stz[2].all[29] := FALSE;   // L1-PROFINET[29]
   linea.stz[2].all[30] := FALSE;   // L1-PROFINET[30]
   linea.stz[2].all[31] := FALSE;   // L1-PROFINET[31]
   linea.stz[2].all[32] := FALSE;   // L1-PROFINET[32]
   linea.stz[2].all[33] := FALSE;   // L1-PROFINET[33]
   linea.stz[2].all[34] := FALSE;   // L1-PROFINET[34]
   linea.stz[2].all[35] := FALSE;   // L1-PROFINET[35]
   linea.stz[2].all[36] := FALSE;   // L1-PROFINET[36]
   linea.stz[2].all[37] := FALSE;   // L1-PROFINET[37]
   linea.stz[2].all[38] := FALSE;   // L1-PROFINET[38]
   linea.stz[2].all[39] := FALSE;   // L1-PROFINET[39]
   linea.stz[2].all[40] := FALSE;   // L1-PROFINET[40]
   linea.stz[2].all[41] := FALSE;   // L1-PROFINET[41]
   linea.stz[2].all[42] := FALSE;   // L1-PROFINET[42]
   linea.stz[2].all[43] := FALSE;   // L1-PROFINET[43]
   linea.stz[2].all[44] := FALSE;   // L1-PROFINET[44]
   linea.stz[2].all[45] := FALSE;   // L1-PROFINET[45]
   linea.stz[2].all[46] := FALSE;   // L1-PROFINET[46]
   linea.stz[2].all[47] := FALSE;   // L1-PROFINET[47]
   linea.stz[2].all[48] := FALSE;   // L1-PROFINET[48]
   linea.stz[2].all[49] := FALSE;   // L1-PROFINET[49]
   linea.stz[2].all[50] := FALSE;   // L1-PROFINET[50]-ERRORE COMUNICAZIONE
   linea.stz[2].all[51] := FALSE;   // L1-PROFINET[51]
   linea.stz[2].all[52] := FALSE;   // L1-PROFINET[52]-ERRORE COMUNICAZIONE
   linea.stz[2].all[53] := FALSE;   // L1-PROFINET[53]
   linea.stz[2].all[54] := FALSE;   // L1-PROFINET[54]-ERRORE COMUNICAZIONE
   linea.stz[2].all[55] := FALSE;   // L1-PROFINET[55]
   linea.stz[2].all[56] := FALSE;   // L1-PROFINET[56]-ERRORE COMUNICAZIONE
   linea.stz[2].all[57] := FALSE;   // L1-PROFINET[57]
   linea.stz[2].all[58] := FALSE;   // L1-PROFINET[58]
   linea.stz[2].all[59] := FALSE;   // L1-PROFINET[59]
   linea.stz[2].all[60] := FALSE;   // L1-PROFINET[60]-ERRORE COMUNICAZIONE
   linea.stz[2].all[61] := FALSE;   // L1-PROFINET[61]-ERRORE COMUNICAZIONE
   linea.stz[2].all[62] := FALSE;   // L1-PROFINET[62]
   linea.stz[2].all[63] := FALSE;   // L1-PROFINET[63]
   linea.stz[2].all[64] := FALSE;   // L1-PROFINET[64]-ERRORE COMUNICAZIONE
   linea.stz[2].all[65] := FALSE;   // L1-PROFINET[65]-ERRORE COMUNICAZIONE
   linea.stz[2].all[66] := FALSE;   // L1-PROFINET[66]-ERRORE COMUNICAZIONE
   linea.stz[2].all[67] := FALSE;   // L1-PROFINET[67]-ERRORE COMUNICAZIONE
   linea.stz[2].all[68] := FALSE;   // L1-PROFINET[68]
   linea.stz[2].all[69] := FALSE;   // L1-PROFINET[69]
   linea.stz[2].all[70] := FALSE;   // L1-PROFINET[70]
   linea.stz[2].all[71] := FALSE;   // L1-PROFINET[71]
   linea.stz[2].all[72] := FALSE;   // L1-PROFINET[72]
   linea.stz[2].all[73] := FALSE;   // L1-PROFINET[73]
   linea.stz[2].all[74] := FALSE;   // L1-PROFINET[74]
   linea.stz[2].all[75] := FALSE;   // L1-PROFINET[75]
   linea.stz[2].all[76] := FALSE;   // L1-PROFINET[76]
   linea.stz[2].all[77] := FALSE;   // L1-PROFINET[77]
   linea.stz[2].all[78] := FALSE;   // L1-PROFINET[78]
   linea.stz[2].all[79] := FALSE;   // L1-PROFINET[79]
   linea.stz[2].all[80] := FALSE;   // L1-PROFINET[80]
   linea.stz[2].all[81] := FALSE;   // L1-PROFINET[81]
   linea.stz[2].all[82] := FALSE;   // L1-PROFINET[82]
   linea.stz[2].all[83] := FALSE;   // L1-PROFINET[83]
   linea.stz[2].all[84] := FALSE;   // L1-PROFINET[84]
   linea.stz[2].all[85] := FALSE;   // L1-PROFINET[85]
   linea.stz[2].all[86] := FALSE;   // L1-PROFINET[86]
   linea.stz[2].all[87] := FALSE;   // L1-PROFINET[87]
   linea.stz[2].all[88] := FALSE;   // L1-PROFINET[88]
   linea.stz[2].all[89] := FALSE;   // L1-PROFINET[89]
   linea.stz[2].all[90] := FALSE;   // L1-PROFINET[90]
   linea.stz[2].all[91] := FALSE;   // L1-PROFINET[91]
   linea.stz[2].all[92] := FALSE;   // L1-PROFINET[92]
   linea.stz[2].all[93] := FALSE;   // L1-PROFINET[93]
   linea.stz[2].all[94] := FALSE;   // L1-PROFINET[94]
   linea.stz[2].all[95] := FALSE;   // L1-PROFINET[95]
   linea.stz[2].all[96] := FALSE;   // L1-PROFINET[96]
   linea.stz[2].all[97] := FALSE;   // L1-PROFINET[97]
   linea.stz[2].all[98] := FALSE;   // L1-PROFINET[98]
   linea.stz[2].all[99] := FALSE;   // L1-PROFINET[99]
   linea.stz[2].all[100] := FALSE;   // L1-PROFINET[100]-ERRORE COMUNICAZIONE
   linea.stz[2].all[101] := FALSE;   // L1-PROFINET[101]
   linea.stz[2].all[102] := FALSE;   // L1-PROFINET[102]-ERRORE COMUNICAZIONE
   linea.stz[2].all[103] := FALSE;   // L1-PROFINET[103]
   linea.stz[2].all[104] := FALSE;   // L1-PROFINET[104]-ERRORE COMUNICAZIONE
   linea.stz[2].all[105] := FALSE;   // L1-PROFINET[105]
   linea.stz[2].all[106] := FALSE;   // L1-PROFINET[106]-ERRORE COMUNICAZIONE
   linea.stz[2].all[107] := FALSE;   // L1-PROFINET[107]
   linea.stz[2].all[108] := FALSE;   // L1-PROFINET[108]-ERRORE COMUNICAZIONE
   linea.stz[2].all[109] := FALSE;   // L1-PROFINET[109]
   linea.stz[2].all[110] := FALSE;   // L1-PROFINET[110]-ERRORE COMUNICAZIONE
   linea.stz[2].all[111] := FALSE;   // L1-PROFINET[111]
   linea.stz[2].all[112] := FALSE;   // L1-PROFINET[112]-ERRORE COMUNICAZIONE
   linea.stz[2].all[113] := FALSE;   // L1-PROFINET[113]
   linea.stz[2].all[114] := FALSE;   // L1-PROFINET[114]-ERRORE COMUNICAZIONE
   linea.stz[2].all[115] := FALSE;   // L1-PROFINET[115]
   linea.stz[2].all[116] := FALSE;   // L1-PROFINET[116]-ERRORE COMUNICAZIONE
   linea.stz[2].all[117] := FALSE;   // L1-PROFINET[117]
   linea.stz[2].all[118] := FALSE;   // L1-PROFINET[118]-ERRORE COMUNICAZIONE
   linea.stz[2].all[119] := FALSE;   // L1-PROFINET[119]
   linea.stz[2].all[120] := FALSE;   // L1-PROFINET[120]-ERRORE COMUNICAZIONE
   linea.stz[2].all[121] := FALSE;   // L1-PROFINET[121]
   linea.stz[2].all[122] := FALSE;   // L1-PROFINET[122]-ERRORE COMUNICAZIONE
   linea.stz[2].all[123] := FALSE;   // L1-PROFINET[123]
   linea.stz[2].all[124] := FALSE;   // L1-PROFINET[124]-ERRORE COMUNICAZIONE
   linea.stz[2].all[125] := FALSE;   // L1-PROFINET[125]
   linea.stz[2].all[126] := FALSE;   // L1-PROFINET[126]-ERRORE COMUNICAZIONE
   linea.stz[2].all[127] := FALSE;   // L1-PROFINET[127]
   linea.stz[2].all[128] := FALSE;   // L1-PROFINET[128]-ERRORE COMUNICAZIONE
   linea.stz[2].all[129] := FALSE;   // L1-PROFINET[129]
   linea.stz[2].all[130] := FALSE;   // L1-PROFINET[130]-ERRORE COMUNICAZIONE
   linea.stz[2].all[131] := FALSE;   // L1-PROFINET[131]
   linea.stz[2].all[132] := FALSE;   // L1-PROFINET[132]-ERRORE COMUNICAZIONE
   linea.stz[2].all[133] := FALSE;   // L1-PROFINET[133]
   linea.stz[2].all[134] := FALSE;   // L1-PROFINET[134]-ERRORE COMUNICAZIONE
   linea.stz[2].all[135] := FALSE;   // L1-PROFINET[135]
   linea.stz[2].all[136] := FALSE;   // L1-PROFINET[136]-ERRORE COMUNICAZIONE
   linea.stz[2].all[137] := FALSE;   // L1-PROFINET[137]
   linea.stz[2].all[138] := FALSE;   // L1-PROFINET[138]-ERRORE COMUNICAZIONE
   linea.stz[2].all[139] := FALSE;   // L1-PROFINET[139]
   linea.stz[2].all[140] := FALSE;   // L1-PROFINET[140]-ERRORE COMUNICAZIONE
   linea.stz[2].all[141] := FALSE;   // L1-PROFINET[141]
   linea.stz[2].all[142] := FALSE;   // L1-PROFINET[142]-ERRORE COMUNICAZIONE
   linea.stz[2].all[143] := FALSE;   // L1-PROFINET[143]
   linea.stz[2].all[144] := FALSE;   // L1-PROFINET[144]-ERRORE COMUNICAZIONE
   linea.stz[2].all[145] := FALSE;   // L1-PROFINET[145]
   linea.stz[2].all[146] := FALSE;   // L1-PROFINET[146]-ERRORE COMUNICAZIONE
   linea.stz[2].all[147] := FALSE;   // L1-PROFINET[147]
   linea.stz[2].all[148] := FALSE;   // L1-PROFINET[148]-ERRORE COMUNICAZIONE
   linea.stz[2].all[149] := FALSE;   // L1-PROFINET[149]
   linea.stz[2].all[150] := FALSE;   // L1-PROFINET[150]-ERRORE COMUNICAZIONE
   linea.stz[2].all[151] := FALSE;   // L1-PROFINET[151]
   linea.stz[2].all[152] := FALSE;   // L1-PROFINET[152]-ERRORE COMUNICAZIONE
   linea.stz[2].all[153] := FALSE;   // L1-PROFINET[153]
   linea.stz[2].all[154] := FALSE;   // L1-PROFINET[154]-ERRORE COMUNICAZIONE
   linea.stz[2].all[155..192] := FALSE;
   linea.stz[3].all[1] := TRUE;   // L1-GENERALE[1]-COMUNICAZIONE PC PLC INTERROTTA
   linea.stz[3].all[2..192] := FALSE;
   linea.stz[4].all[1] := FALSE;   // L1-ASPO[1]-24-L411+-LINEA NON RIPRISTINATA
   linea.stz[4].all[2] := TRUE;   // L1-ASPO[1]-24-L412+-LINEA NON RIPRISTINATA
   linea.stz[4].all[3] := FALSE;   // L1-ASPO[3]-AUTOMATICO CON BRACCIO PREMICOIL BASSO
   linea.stz[4].all[4] := FALSE;   // L1-ASPO[4]- SVOLGITORE GTA MINIMA PRESSIONE
   linea.stz[4].all[5] := FALSE;   // L1-ASPO[5]-M101 MADRINO -FAULT DATI SETTING
   linea.stz[4].all[6] := FALSE;   // L1-ASPO[6]-M101 MADRINO -FAULT DATI MACCHINA
   linea.stz[4].all[7] := FALSE;   // L1-ASPO[7]-M101 MADRINO -ANSA ALTA
   linea.stz[4].all[8] := FALSE;   // L1-ASPO[8]
   linea.stz[4].all[9] := FALSE;   // L1-ASPO[9]-M101 MADRINO -FAULT DRIVE
   linea.stz[4].all[10] := FALSE;   // L1-ASPO[10]-M101 MADRINO -PROTEZIONE FRENO INTERVENUTA
   linea.stz[4].all[11] := FALSE;   // L1-ASPO[11]-M101 MADRINO -PROTEZIONE VENTILATORI
   linea.stz[4].all[12] := FALSE;   // L1-ASPO[12]-M101 MADRINO -FAULT
   linea.stz[4].all[13] := FALSE;   // L1-ASPO[13]-M101 MADRINO -BRACCIO PREMICOIL NON IN POSIZIONE
   linea.stz[4].all[14] := FALSE;   // L1-ASPO[14]
   linea.stz[4].all[15] := FALSE;   // L1-ASPO[15]-CENTRALE OLEODINAMICA-PROTEZIONE INTERVENUTA
   linea.stz[4].all[16] := FALSE;   // L1-ASPO[16]-CENTRALE OLEODINAMICA-ALLARME TEMPERATURA
   linea.stz[4].all[17] := FALSE;   // L1-ASPO[17]-CENTRALE OLEODINAMICA-SUPERATO TEMPO MASSIMO LAVORO
   linea.stz[4].all[18] := FALSE;   // L1-ASPO[18]-CENTRALE OLEODINAMICA-MINIMO LIVELLO OLIO
   linea.stz[4].all[19] := FALSE;   // L1-ASPO[19]
   linea.stz[4].all[20] := FALSE;   // L1-ASPO[20]-H401- ANOMALIA MOVIMENTO 1 SPOOL VALVOLA ESPANSIONE MANDRINO 1
   linea.stz[4].all[21] := FALSE;   // L1-ASPO[21]-H401- ANOMALIA MOVIMENTO 2 SPOOL VALVOLA CONTRAZIONE MANDRINO 1
   linea.stz[4].all[22] := FALSE;   // L1-ASPO[22]-
   linea.stz[4].all[23] := FALSE;   // L1-ASPO[23]-
   linea.stz[4].all[24] := FALSE;   // L1-ASPO[24]
   linea.stz[4].all[25] := FALSE;   // L1-ASPO[25]-H402- ANOMALIA MOVIMENTO 1 SPOOL VALVOLA ESPANSIONE MANDRINO 2
   linea.stz[4].all[26] := FALSE;   // L1-ASPO[26]-H402- ANOMALIA MOVIMENTO 2 SPOOL VALVOLA CONTRAZIONE MANDRINO 2
   linea.stz[4].all[27] := FALSE;   // L1-ASPO[27]-H402-
   linea.stz[4].all[28] := FALSE;   // L1-ASPO[28]-H402-
   linea.stz[4].all[29] := FALSE;   // L1-ASPO[29]
   linea.stz[4].all[30] := FALSE;   // L1-ASPO[30]- DIAMETRO COIL-ANOMALIA LASER LETTURA
   linea.stz[4].all[31] := FALSE;   // L1-ASPO[31]- ANSA XC142A-1-ANOMALIA LASER LETTURA
   linea.stz[4].all[32] := FALSE;   // L1-ASPO[32]- ANSA XC142A-2-ANOMALIA LASER LETTURA
   linea.stz[4].all[33..35] := FALSE;
   linea.stz[4].all[36] := FALSE;   // L1-ASPO[36]-M102 MADRINO -FAULT DATI SETTING
   linea.stz[4].all[37] := FALSE;   // L1-ASPO[37]-M102 MADRINO -FAULT DATI MACCHINA
   linea.stz[4].all[38..39] := FALSE;
   linea.stz[4].all[40] := FALSE;   // L1-ASPO[40]-M102 MADRINO -FAULT DRIVE
   linea.stz[4].all[41] := FALSE;   // L1-ASPO[41]-M102 MADRINO -PROTEZIONE FRENO INTERVENUTA
   linea.stz[4].all[42] := FALSE;   // L1-ASPO[42]-M102 MADRINO -PROTEZIONE VENTILATORI
   linea.stz[4].all[43] := FALSE;   // L1-ASPO[43]-M102 MADRINO -FAULT
   linea.stz[4].all[44] := FALSE;   // L1-ASPO[44]-M102 MADRINO -BRACCIO PREMICOIL NON IN POSIZIONE
   linea.stz[4].all[45..49] := FALSE;
   linea.stz[4].all[50] := FALSE;   // L1-ASPO[50]-YVA14.2 ANOMALIA MOVIMENTO 1 SPOOL VALVOLA SEZIONATRICE MANDRINO 1
   linea.stz[4].all[51] := FALSE;   // L1-ASPO[51]-YVA14.2 ANOMALIA MOVIMENTO 2 SPOOL VALVOLA SEZIONATRICE MANDRINO 2
   linea.stz[4].all[52] := FALSE;   // L1-ASPO[52]-YVA14.3 ANOMALIA MOVIMENTO 1 SPOOL VALVOLA SEZIONATRICE MANDRINO 2
   linea.stz[4].all[53] := FALSE;   // L1-ASPO[53]-YVA14.3 ANOMALIA MOVIMENTO 2 SPOOL VALVOLA SEZIONATRICE MANDRINO 2
   linea.stz[4].all[54] := FALSE;   // L1-ASPO[54]-YVA14.1 ANOMALIA MOVIMENTO 1 SPOOL VALVOLA SEZIONATRICE TIN
   linea.stz[4].all[55] := FALSE;   // L1-ASPO[55]-YVA14.1 ANOMALIA MOVIMENTO 2 SPOOL VALVOLA SEZIONATRICE TIN
   linea.stz[4].all[56..59] := FALSE;
   linea.stz[4].all[60] := FALSE;   // L1-ASPO[60]-M112 TORRETTA -FAULT DRIVE
   linea.stz[4].all[61] := FALSE;   // L1-ASPO[61]-M112 TORRETTA -PROTEZIONE FRENO INTERVENUTA
   linea.stz[4].all[62] := FALSE;   // L1-ASPO[62]-M112 TORRETTA -PROTEZIONE VENTILATORI
   linea.stz[4].all[63] := FALSE;   // L1-ASPO[63]-M112 TORRETTA -FAULT
   linea.stz[4].all[64] := FALSE;   // L1-ASPO[64]-M112 TORRETTA -PRESENZA LAMIERA SU RADDRIZZATRICE
   linea.stz[4].all[65..69] := FALSE;
   linea.stz[4].all[70] := FALSE;   // L1-ASPO[70]-H407 TIMEOUT MOVIMENTO NEGATIVO SALITA/DISCESA TIN
   linea.stz[4].all[71] := FALSE;   // L1-ASPO[71]-H408 TIMEOUT MOVIMENTO CONTRAZIONE/ESPANSIONE TIN
   linea.stz[4].all[72] := FALSE;   // L1-ASPO[72]-H409 TIMEOUT MOVIMENTO SALITA/DISCESA DEFLETTORE TIN
   linea.stz[4].all[73..192] := FALSE;
   linea.stz[5].all[1] := FALSE;   // L1-RADDRIZZATRICE[1]
   linea.stz[5].all[2] := FALSE;   // L1-RADDRIZZATRICE[2]
   linea.stz[5].all[3] := FALSE;   // L1-RADDRIZZATRICE[3]
   linea.stz[5].all[4] := FALSE;   // L1-RADDRIZZATRICE[4]
   linea.stz[5].all[5] := FALSE;   // L1-RADDRIZZATRICE[5]-M141-FAULT DRIVE
   linea.stz[5].all[6] := FALSE;   // L1-RADDRIZZATRICE[6]-M141-PROTEZIONE FRENO INTERVENUTA
   linea.stz[5].all[7] := FALSE;   // L1-RADDRIZZATRICE[7]-M141-PROTEZIONE VENTILATORI
   linea.stz[5].all[8] := FALSE;   // L1-RADDRIZZATRICE[8]-M141-FAULT
   linea.stz[5].all[9] := FALSE;   // L1-RADDRIZZATRICE[9]
   linea.stz[5].all[10] := FALSE;   // L1-RADDRIZZATRICE[10]-P501-PINCHROLL-TIMEOUT MOVIMENTO POSITIVO
   linea.stz[5].all[11] := FALSE;   // L1-RADDRIZZATRICE[11]-P501-PINCHROLL-TIMEOUT MOVIMENTO NEGATIVO
   linea.stz[5].all[12] := FALSE;   // L1-RADDRIZZATRICE[12]-P501-PINCHROLL-MOVIMENTO NON POSSIBILE
   linea.stz[5].all[13] := FALSE;   // L1-RADDRIZZATRICE[13]-P501-PINCHROLL-NON IN POSIZIONE PER START CICLO
   linea.stz[5].all[14] := FALSE;   // L1-RADDRIZZATRICE[14]
   linea.stz[5].all[15] := FALSE;   // L1-RADDRIZZATRICE[15]-M141-FAULT DATI SETTING
   linea.stz[5].all[16] := FALSE;   // L1-RADDRIZZATRICE[16]-M141-FAULT DATI MACCHINA
   linea.stz[5].all[17] := FALSE;   // L1-RADDRIZZATRICE[17]-M141-TAVOLA ACCOMPAGNAMENTO FUORI POSIZIONE
   linea.stz[5].all[18] := FALSE;   // L1-RADDRIZZATRICE[18]-M141-ANSA ALTA
   linea.stz[5].all[19] := FALSE;   // L1-RADDRIZZATRICE[19]-M141-MINIMA PRESSIONE ARIA
   linea.stz[5].all[20] := FALSE;   // L1-RADDRIZZATRICE[20]
   linea.stz[5].all[21] := FALSE;   // L1-RADDRIZZATRICE[21]-LASER 1 ANSA-ANOMALIA LASER LETTURA
   linea.stz[5].all[22] := FALSE;   // L1-RADDRIZZATRICE[22]-LASER 2 ANSA-ANOMALIA LASER LETTURA
   linea.stz[5].all[23..29] := FALSE;
   linea.stz[5].all[30] := FALSE;   // L1-RADDRIZZATRICE[30]-P501 TIMEOUT MOVIMENTO POSITIVO
   linea.stz[5].all[31] := FALSE;   // L1-RADDRIZZATRICE[31]-P501 TIMEOUT MOVIMENTO NEGATIVO
   linea.stz[5].all[32] := FALSE;   // L1-RADDRIZZATRICE[32]-P501 MOVIMENTO NON POSSIBILE
   linea.stz[5].all[33..39] := FALSE;
   linea.stz[5].all[40] := FALSE;   // L1-RADDRIZZATRICE[40]-M140 FAULT DRIVE
   linea.stz[5].all[41] := FALSE;   // L1-RADDRIZZATRICE[41]-M140 FAULT DATI MACCHINA
   linea.stz[5].all[42] := FALSE;   // L1-RADDRIZZATRICE[42]-M140 FINECORSA SOFTWARE NEGATIVO
   linea.stz[5].all[43] := FALSE;   // L1-RADDRIZZATRICE[43]-M140 FINECORSA SOFTWARE POSITIVO
   linea.stz[5].all[44] := FALSE;   // L1-RADDRIZZATRICE[44]-M140 FINECORSA NEGATIVO
   linea.stz[5].all[45] := FALSE;   // L1-RADDRIZZATRICE[45]-M140 FINECORSA POSITIVO
   linea.stz[5].all[46] := FALSE;   // L1-RADDRIZZATRICE[46]-M140 ALLARME TERMICO
   linea.stz[5].all[47..48] := FALSE;
   linea.stz[5].all[49] := FALSE;   // L1-RADDRIZZATRICE[49]-M141 MOTORE INSERITO - AUTOMATICO NON POSSIBILE
   linea.stz[5].all[50..192] := FALSE;
   linea.stz[6].all[1] := FALSE;   // L1-GIUNZIONE[1]-24-L42+-LINEA NON RIPRISTINATA
   linea.stz[6].all[2] := FALSE;   // L1-GIUNZIONE[2]
   linea.stz[6].all[3] := FALSE;   // L1-GIUNZIONE[3]
   linea.stz[6].all[4] := FALSE;   // L1-GIUNZIONE[4]
   linea.stz[6].all[5] := FALSE;   // L1-GIUNZIONE[5]-H601 -CESOIA GIUNZIONE-TIMEOUT MOVIMENTO POSITIVO
   linea.stz[6].all[6] := FALSE;   // L1-GIUNZIONE[6]-H601 -CESOIA GIUNZIONE-TIMEOUT MOVIMENTO NEGATIVO
   linea.stz[6].all[7] := FALSE;   // L1-GIUNZIONE[7]-H601 -CESOIA GIUNZIONE-MOVIMENTO NON POSSIBILE
   linea.stz[6].all[8] := FALSE;   // L1-GIUNZIONE[8]-H601 -CESOIA GIUNZIONE-NON IN POSIZIONE PER START CICLO
   linea.stz[6].all[9] := FALSE;   // L1-GIUNZIONE[9]
   linea.stz[6].all[10] := FALSE;   // L1-GIUNZIONE[10]-CENTRALE OLEODINAMICA-PROTEZIONE INTERVENUTA
   linea.stz[6].all[11] := FALSE;   // L1-GIUNZIONE[11]-CENTRALE OLEODINAMICA-MASSIMA TEMPERATURA
   linea.stz[6].all[12] := FALSE;   // L1-GIUNZIONE[12]-CENTRALE OLEODINAMICA-SUPERATO TEMPO MASSIMO LAVORO
   linea.stz[6].all[13] := FALSE;   // L1-GIUNZIONE[13]-CENTRALE OLEODINAMICA-MINIMO LIVELLO OLIO
   linea.stz[6].all[14] := FALSE;   // L1-GIUNZIONE[14]
   linea.stz[6].all[15] := FALSE;   // L1-GIUNZIONE[15]-H601 -CESOIA GIUNZIONE-PERNO DI BLOCCAGGIO INSERITO
   linea.stz[6].all[16] := FALSE;   // L1-GIUNZIONE[16]-H601 -CESOIA GIUNZIONE-MORSE NON APERTE
   linea.stz[6].all[17..192] := FALSE;
   linea.stz[7].all[1] := FALSE;   // L1-ALIM + PUNZ[1]
   linea.stz[7].all[2] := FALSE;   // L1-ALIM + PUNZ[2]
   linea.stz[7].all[3] := FALSE;   // L1-ALIM + PUNZ[3]
   linea.stz[7].all[4] := FALSE;   // L1-ALIM + PUNZ[4]
   linea.stz[7].all[5] := FALSE;   // L1-ALIM + PUNZ[5]-M201-ALIMENTATORE A RULLI-FAULT DRIVE
   linea.stz[7].all[6] := FALSE;   // L1-ALIM + PUNZ[6]-M201-ALIMENTATORE A RULLI-PROTEZIONE VENTILATORI
   linea.stz[7].all[7] := FALSE;   // L1-ALIM + PUNZ[7]-M201-ALIMENTATORE A RULLI-MOVIMENTO NON POSSIBILE
   linea.stz[7].all[8] := FALSE;   // L1-ALIM + PUNZ[8]-M201-ALIMENTATORE A RULLI-FAULT
   linea.stz[7].all[9] := FALSE;   // L1-ALIM + PUNZ[9]-P701-SALITA DISCESA ALIMENTATORE-TIMEOUT MOVIMENTO POSITIVO
   linea.stz[7].all[10] := FALSE;   // L1-ALIM + PUNZ[10]-P701-SALITA DISCESA ALIMENTATORE-TIMEOUT MOVIMENTO NEGATIVO
   linea.stz[7].all[11] := FALSE;   // L1-ALIM + PUNZ[11]-P701-SALITA DISCESA ALIMENTATORE-MOVIMENTO NON POSSIBILE
   linea.stz[7].all[12] := FALSE;   // L1-ALIM + PUNZ[12]-P701-SALITA DISCESA ALIMENTATORE-NON IN POSIZIONE PER START CICLO
   linea.stz[7].all[13] := FALSE;   // L1-ALIM + PUNZ[13]-P01-01 CASSETTO-TIMEOUT MOVIMENTO POSITIVO
   linea.stz[7].all[14] := FALSE;   // L1-ALIM + PUNZ[14]-P01-01 CASSETTO-TIMEOUT MOVIMENTO NEGATIVO
   linea.stz[7].all[15] := FALSE;   // L1-ALIM + PUNZ[15]-P01-01 CASSETTO-MOVIMENTO NON POSSIBILE
   linea.stz[7].all[16] := FALSE;   // L1-ALIM + PUNZ[16]-P01-01 CASSETTO-NON IN POSIZIONE PER START CICLO
   linea.stz[7].all[17] := FALSE;   // L1-ALIM + PUNZ[17]
   linea.stz[7].all[18] := FALSE;   // L1-ALIM + PUNZ[18]-FINE PRODUZIONE
   linea.stz[7].all[19] := FALSE;   // L1-ALIM + PUNZ[19]-PREAVVISO FINE PRODUZIONE
   linea.stz[7].all[20] := FALSE;   // L1-ALIM + PUNZ[20]
   linea.stz[7].all[21] := FALSE;   // L1-ALIM + PUNZ[21]-PRESSA-ERRORE ENCODER CON PMS
   linea.stz[7].all[22] := FALSE;   // L1-ALIM + PUNZ[22]-PRESSA-FAULT
   linea.stz[7].all[23] := FALSE;   // L1-ALIM + PUNZ[23]-PRESSA-MODALITA DI LAVORO NON CORRETTA
   linea.stz[7].all[24] := FALSE;   // L1-ALIM + PUNZ[24]-PRESSA-PRESSA NON AL PMS
   linea.stz[7].all[25] := FALSE;   // L1-ALIM + PUNZ[25]-PRESSA-PASSO ALIMENTATORE NON ESEGUITO
   linea.stz[7].all[26] := FALSE;   // L1-ALIM + PUNZ[26]-PRESSA-CASSETTI STAMPO NON IN POSIZIONE
   linea.stz[7].all[27] := FALSE;   // L1-ALIM + PUNZ[27]-PRESSA-FAULT DATI MACCHINA
   linea.stz[7].all[28] := FALSE;   // L1-ALIM + PUNZ[28]-ANSA ALTA
   linea.stz[7].all[29] := FALSE;   // L1-ALIM + PUNZ[29]-LASER 1 ANSA-ANOMALIA LASER LETTURA
   linea.stz[7].all[30] := FALSE;   // L1-ALIM + PUNZ[30]-LASER 2 ANSA-ANOMALIA LASER LETTURA
   linea.stz[7].all[31] := FALSE;   // L1-ALIM + PUNZ[31]-TAVOLA ACCOMPAGNAMENTO FUORI POSIZIONE
   linea.stz[7].all[32] := FALSE;   // L1-ALIM + PUNZ[32]-LISTA COMPILATA MOVIMENTO NON POSSIBILE
   linea.stz[7].all[33] := FALSE;   // L1-ALIM + PUNZ[33]-M201-ALIMENTATORE A RULLI-NON IN POSIZIONE PER START CICLO
   linea.stz[7].all[34] := FALSE;   // L1-ALIM + PUNZ[34]-AUTOMATICO CON LISTA NON COMPILATA
   linea.stz[7].all[35] := FALSE;   // L1-ALIM + PUNZ[35]-DROPSA-MINIMO LIVELLO OLIO
   linea.stz[7].all[36] := FALSE;   // L1-ALIM + PUNZ[36]-DROPSA-MANCATA LUBRIFICAZIONE
   linea.stz[7].all[37..192] := FALSE;
   linea.stz[8].all[1] := FALSE;   // L1-PROFILA[1]-24-L43+-LINEA NON RIPRISTINATA
   linea.stz[8].all[2] := FALSE;   // L1-PROFILA[2] - MINIMA PRESSIONE ARIA GTA
   linea.stz[8].all[3] := FALSE;   // L1-PROFILA[3]
   linea.stz[8].all[4] := FALSE;   // L1-PROFILA[4]
   linea.stz[8].all[5] := FALSE;   // L1-PROFILA[5]-M301 PROFILA-FAULT DRIVE
   linea.stz[8].all[6] := FALSE;   // L1-PROFILA[6]-M301 PROFILA-PROTEZIONE FRENO INTERVENUTA
   linea.stz[8].all[7] := FALSE;   // L1-PROFILA[7]-M301 PROFILA-PROTEZIONE VENTILATORI
   linea.stz[8].all[8] := FALSE;   // L1-PROFILA[8]-M301 PROFILA-FAULT
   linea.stz[8].all[9] := FALSE;   // L1-PROFILA[9]-M365 ESTRATTORE-FAULT DRIVE
   linea.stz[8].all[10] := FALSE;   // L1-PROFILA[10]-M365 ESTRATTORE-PROTEZIONE FRENO INTERVENUTA
   linea.stz[8].all[11] := FALSE;   // L1-PROFILA[11]-M365 ESTRATTORE-TIMEOUT MOVIMENTO POSITIVO
   linea.stz[8].all[12] := FALSE;   // L1-PROFILA[12]-M365 ESTRATTORE-FAULT
   linea.stz[8].all[13] := FALSE;   // L1-PROFILA[13]
   linea.stz[8].all[14] := FALSE;   // L1-PROFILA[14]-P801 RUOTA METRICA-TIMEOUT MOVIMENTO POSITIVO
   linea.stz[8].all[15] := FALSE;   // L1-PROFILA[15]-P801 RUOTA METRICA-TIMEOUT MOVIMENTO NEGATIVO
   linea.stz[8].all[16] := FALSE;   // L1-PROFILA[16]-P801 RUOTA METRICA-MOVIMENTO NON POSSIBILE
   linea.stz[8].all[17] := FALSE;   // L1-PROFILA[17]-P801 RUOTA METRICA-NON IN POSIZIONE PER START CICLO
   linea.stz[8].all[18] := FALSE;   // L1-PROFILA[18]
   linea.stz[8].all[19] := FALSE;   // L1-PROFILA[19]
   linea.stz[8].all[20] := FALSE;   // L1-PROFILA[20]-SALDATRICE-ERRORE COMUNICAZIONE
   linea.stz[8].all[21] := FALSE;
   linea.stz[8].all[22] := FALSE;   // L1-PROFILA[22]-LUBRIFICAZIONE-MINIMO LIVELLO OLIO
   linea.stz[8].all[23..55] := FALSE;
   linea.stz[8].all[56] := TRUE;
   linea.stz[8].all[57..65] := FALSE;
   linea.stz[8].all[66] := TRUE;
   linea.stz[8].all[67..75] := FALSE;
   linea.stz[8].all[76] := TRUE;
   linea.stz[8].all[77..192] := FALSE;
   linea.stz[9].all[1] := FALSE;   // L1-TAGLIO[1]-24-L44+-LINEA NON RIPRISTINATA
   linea.stz[9].all[2] := FALSE;   // L1-TAGLIO[2]
   linea.stz[9].all[3] := FALSE;   // L1-TAGLIO[3]
   linea.stz[9].all[4] := FALSE;   // L1-TAGLIO[4]
   linea.stz[9].all[5] := FALSE;   // L1-TAGLIO[5]
   linea.stz[9].all[6] := FALSE;   // L1-TAGLIO[6]
   linea.stz[9].all[7] := FALSE;   // L1-TAGLIO[7]
   linea.stz[9].all[8] := FALSE;   // L1-TAGLIO[8]
   linea.stz[9].all[9] := FALSE;   // L1-TAGLIO[9]
   linea.stz[9].all[10] := FALSE;   // L1-TAGLIO[10]-M404 SALITA DISCESA DISCO TAGLIO-FAULT DRIVE
   linea.stz[9].all[11] := FALSE;   // L1-TAGLIO[11]-M404 SALITA DISCESA DISCO TAGLIO-PROTEZIONE VENTILATORI
   linea.stz[9].all[12] := FALSE;   // L1-TAGLIO[12]-M404 SALITA DISCESA DISCO TAGLIO-MOVIMENTO NON POSSIBILE
   linea.stz[9].all[13] := FALSE;   // L1-TAGLIO[13]-M404 SALITA DISCESA DISCO TAGLIO-ASSE NON REFERENZIATO
   linea.stz[9].all[14] := FALSE;   // L1-TAGLIO[14]-M404 SALITA DISCESA DISCO TAGLIO-FAULT
   linea.stz[9].all[15] := FALSE;   // L1-TAGLIO[15]-M405 ROTAZIONE DISCO TAGLIO-FAULT DRIVE
   linea.stz[9].all[16] := FALSE;   // L1-TAGLIO[16]-M405 ROTAZIONE DISCO TAGLIO-PROTEZIONE FRENO INTERVENUTA
   linea.stz[9].all[17] := FALSE;   // L1-TAGLIO[17]-M405 ROTAZIONE DISCO TAGLIO-PROTEZIONE VENTILATORI
   linea.stz[9].all[18] := FALSE;   // L1-TAGLIO[18]-M405 ROTAZIONE DISCO TAGLIO-FAULT
   linea.stz[9].all[19] := FALSE;   // L1-TAGLIO[19]-M408 TAPPETO EVACUAZIONE-FAULT DRIVE
   linea.stz[9].all[20] := FALSE;   // L1-TAGLIO[20]-M408 TAPPETO EVACUAZIONE-PROTEZIONE FRENO INTERVENUTA
   linea.stz[9].all[21] := FALSE;   // L1-TAGLIO[21]-M408 TAPPETO EVACUAZIONE-PROTEZIONE VENTILATORI
   linea.stz[9].all[22] := FALSE;   // L1-TAGLIO[22]-M408 TAPPETO EVACUAZIONE-FAULT
   linea.stz[9].all[23] := FALSE;   // L1-TAGLIO[23]-P901 PRESSORE PROFILO-TIMEOUT MOVIMENTO POSITIVO
   linea.stz[9].all[24] := FALSE;   // L1-TAGLIO[24]-P901 PRESSORE PROFILO-TIMEOUT MOVIMENTO NEGATIVO
   linea.stz[9].all[25] := FALSE;   // L1-TAGLIO[25]-P901 PRESSORE PROFILO-MOVIMENTO NON POSSIBILE
   linea.stz[9].all[26] := FALSE;   // L1-TAGLIO[26]-P901 PRESSORE PROFILO-NON IN POSIZIONE PER START CICLO
   linea.stz[9].all[27] := FALSE;   // L1-TAGLIO[27]-P902 MORSE INGRESSO-TIMEOUT MOVIMENTO POSITIVO
   linea.stz[9].all[28] := FALSE;   // L1-TAGLIO[28]-P902 MORSE INGRESSO-TIMEOUT MOVIMENTO NEGATIVO
   linea.stz[9].all[29] := FALSE;   // L1-TAGLIO[29]-P902 MORSE INGRESSO-MOVIMENTO NON POSSIBILE
   linea.stz[9].all[30] := FALSE;   // L1-TAGLIO[30]-P902 MORSE INGRESSO-NON IN POSIZIONE PER START CICLO
   linea.stz[9].all[31] := FALSE;   // L1-TAGLIO[31]-P903 MORSE USCITA-TIMEOUT MOVIMENTO POSITIVO
   linea.stz[9].all[32] := FALSE;   // L1-TAGLIO[32]-P903 MORSE USCITA-TIMEOUT MOVIMENTO NEGATIVO
   linea.stz[9].all[33] := FALSE;   // L1-TAGLIO[33]-P903 MORSE USCITA-MOVIMENTO NON POSSIBILE
   linea.stz[9].all[34] := FALSE;   // L1-TAGLIO[34]-P903 MORSE USCITA-NON IN POSIZIONE PER START CICLO
   linea.stz[9].all[35] := FALSE;   // L1-TAGLIO[35]
   linea.stz[9].all[36] := FALSE;   // L1-TAGLIO[36]-M404 SALITA DISCESA DISCO TAGLIO-FAULT DATI SETTING
   linea.stz[9].all[37] := FALSE;   // L1-TAGLIO[37]-M405 ROTAZIONE DISCO TAGLIO-FAULT DATI SETTING
   linea.stz[9].all[38] := FALSE;   // L1-TAGLIO[38]
   linea.stz[9].all[39] := FALSE;   // L1-TAGLIO[39]
   linea.stz[9].all[40] := FALSE;   // L1-TAGLIO[40]-M401 CARRO TAGLIO AL VOLO-ERRORE COMUNICAZIONE
   linea.stz[9].all[41] := FALSE;   // L1-TAGLIO[41]-M401 CARRO TAGLIO AL VOLO-MODO PARAMETRI ATTIVO
   linea.stz[9].all[42] := FALSE;   // L1-TAGLIO[42]-M401 CARRO TAGLIO AL VOLO-FINECORSA POSITIVO
   linea.stz[9].all[43] := FALSE;   // L1-TAGLIO[43]-M401 CARRO TAGLIO AL VOLO-FINECORSA NEGATIVO
   linea.stz[9].all[44] := FALSE;   // L1-TAGLIO[44]-M401 CARRO TAGLIO AL VOLO-FAULT DRIVE
   linea.stz[9].all[45] := FALSE;   // L1-TAGLIO[45]-M401 CARRO TAGLIO AL VOLO-RESISTENZA DI FRENATURA
   linea.stz[9].all[46] := FALSE;   // L1-TAGLIO[46]-M401 CARRO TAGLIO AL VOLO-PROTEZIONE VENTILATORI
   linea.stz[9].all[47] := FALSE;   // L1-TAGLIO[47]-M401 CARRO TAGLIO AL VOLO-PROGRAMMA NON VALIDO SU SMC
   linea.stz[9].all[48] := FALSE;   // L1-TAGLIO[48]-M401 CARRO TAGLIO AL VOLO-ERRORE GENERICO TAGLIO AL VOLO
   linea.stz[9].all[49] := FALSE;   // L1-TAGLIO[49]-M401 CARRO TAGLIO AL VOLO-CENTRALE IDRAULICA NON OK
   linea.stz[9].all[50] := FALSE;   // L1-TAGLIO[50]-M401 CARRO TAGLIO AL VOLO-CARRO NON IN POSIZIONE DI HOME
   linea.stz[9].all[51] := FALSE;   // L1-TAGLIO[51]-M401 CARRO TAGLIO AL VOLO-MOVIMENTI DI JOG NON POSSIBILI, STAMPO NON APERTO
   linea.stz[9].all[52] := FALSE;   // L1-TAGLIO[52]-M401 CARRO TAGLIO AL VOLO-FAULT
   linea.stz[9].all[53] := FALSE;   // L1-TAGLIO[53]
   linea.stz[9].all[54] := FALSE;   // L1-TAGLIO[54]
   linea.stz[9].all[55] := FALSE;   // L1-TAGLIO[55]-LUNGHEZZA ERRATA
   linea.stz[9].all[56] := FALSE;   // L1-TAGLIO[56]-TIMEOUT CICLO
   linea.stz[9].all[57..59] := FALSE;
   linea.stz[9].all[60] := FALSE;   // L1-TAGLIO[60]-LUBRIFICAZIONE-MINIMO LIVELLO OLIO
   linea.stz[9].all[61..192] := FALSE;
   linea.stz[10].all[1] := FALSE;   // L1-SCARICO[1]
   linea.stz[10].all[2] := FALSE;   // L1-SCARICO[2]
   linea.stz[10].all[3] := FALSE;   // L1-SCARICO[3]
   linea.stz[10].all[4] := FALSE;   // L1-SCARICO[4]
   linea.stz[10].all[5] := FALSE;   // L1-SCARICO[5]-P1001 BANCO SCARICO 1-TIMEOUT MOVIMENTO POSITIVO
   linea.stz[10].all[6] := FALSE;   // L1-SCARICO[6]-P1001 BANCO SCARICO 1-TIMEOUT MOVIMENTO NEGATIVO
   linea.stz[10].all[7] := FALSE;   // L1-SCARICO[7]-P1001 BANCO SCARICO 1-MOVIMENTO NON POSSIBILE
   linea.stz[10].all[8] := FALSE;   // L1-SCARICO[8]-P1001 BANCO SCARICO 1-NON IN POSIZIONE PER START CICLO
   linea.stz[10].all[9] := FALSE;   // L1-SCARICO[9]-P1002 BANCO SCARICO 2-TIMEOUT MOVIMENTO POSITIVO
   linea.stz[10].all[10] := FALSE;   // L1-SCARICO[10]-P1002 BANCO SCARICO 2-TIMEOUT MOVIMENTO NEGATIVO
   linea.stz[10].all[11] := FALSE;   // L1-SCARICO[11]-P1002 BANCO SCARICO 2-MOVIMENTO NON POSSIBILE
   linea.stz[10].all[12] := FALSE;   // L1-SCARICO[12]-P1002 BANCO SCARICO 2-NON IN POSIZIONE PER START CICLO
   linea.stz[10].all[13] := FALSE;   // L1-SCARICO[13]-P1003 BANCO SCARICO 3-TIMEOUT MOVIMENTO POSITIVO
   linea.stz[10].all[14] := FALSE;   // L1-SCARICO[14]-P1003 BANCO SCARICO 3-TIMEOUT MOVIMENTO NEGATIVO
   linea.stz[10].all[15] := FALSE;   // L1-SCARICO[15]-P1003 BANCO SCARICO 3-MOVIMENTO NON POSSIBILE
   linea.stz[10].all[16] := FALSE;   // L1-SCARICO[16]-P1003 BANCO SCARICO 3-NON IN POSIZIONE PER START CICLO
   linea.stz[10].all[17] := FALSE;   // L1-SCARICO[17]-P1004 BANCO SCARICO 4-TIMEOUT MOVIMENTO POSITIVO
   linea.stz[10].all[18] := FALSE;   // L1-SCARICO[18]-P1004 BANCO SCARICO 4-TIMEOUT MOVIMENTO NEGATIVO
   linea.stz[10].all[19] := FALSE;   // L1-SCARICO[19]-P1004 BANCO SCARICO 4-MOVIMENTO NON POSSIBILE
   linea.stz[10].all[20] := FALSE;   // L1-SCARICO[20]-P1004 BANCO SCARICO 4-NON IN POSIZIONE PER START CICLO
   linea.stz[10].all[21] := FALSE;   // L1-SCARICO[21]
   linea.stz[10].all[22] := FALSE;   // L1-SCARICO[22]-RIMUOVERE SCARTO
   linea.stz[10].all[23..192] := FALSE;
   linea.stz[11].all[1..192] := FALSE;
   linea.stz[12].all[1..192] := FALSE;
   linea.stz[13].all[1..192] := FALSE;
   linea.stz[14].all[1..192] := FALSE;
   linea.stz[15].all[1..192] := FALSE;
   linea.stz[16].all[1..192] := FALSE;
   linea.stz[17].all[1..192] := FALSE;
   linea.stz[18].all[1..192] := FALSE;
   linea.stz[19].all[1..192] := FALSE;
   linea.stz[20].all[1..192] := FALSE;
   linea.stz[1].allarmipc[1..6] := 0;
   linea.stz[2].allarmipc[1..6] := 0;
   linea.stz[3].allarmipc[1] := 1;
   linea.stz[3].allarmipc[2..6] := 0;
   linea.stz[4].allarmipc[1] := 2;
   linea.stz[4].allarmipc[2..6] := 0;
   linea.stz[5].allarmipc[1..6] := 0;
   linea.stz[6].allarmipc[1..6] := 0;
   linea.stz[7].allarmipc[1..6] := 0;
   linea.stz[8].allarmipc[1] := 0;
   linea.stz[8].allarmipc[2] := 8388608;
   linea.stz[8].allarmipc[3] := 2050;
   linea.stz[8].allarmipc[4..6] := 0;
   linea.stz[9].allarmipc[1..6] := 0;
   linea.stz[10].allarmipc[1..6] := 0;
   linea.stz[11].allarmipc[1..6] := 0;
   linea.stz[12].allarmipc[1..6] := 0;
   linea.stz[13].allarmipc[1..6] := 0;
   linea.stz[14].allarmipc[1..6] := 0;
   linea.stz[15].allarmipc[1..6] := 0;
   linea.stz[16].allarmipc[1..6] := 0;
   linea.stz[17].allarmipc[1..6] := 0;
   linea.stz[18].allarmipc[1..6] := 0;
   linea.stz[19].allarmipc[1..6] := 0;
   linea.stz[20].allarmipc[1..6] := 0;
   linea.stz[1].war[1..32] := FALSE;
   linea.stz[2].war[1..32] := FALSE;
   linea.stz[3].war[1..32] := FALSE;
   linea.stz[4].war[1..4] := FALSE;
   linea.stz[4].war[5] := FALSE;   // L1-ASPO[5]-M101 MADRINO -PRESENZA LAMIERA
   linea.stz[4].war[6] := TRUE;   // L1-ASPO[6]-CENTRALE OLEODINAMICA-MINIMO LIVELLO OLIO
   linea.stz[4].war[7] := FALSE;   // L1-ASPO[7]-ESPANSIONE MANDRINO-FUNZIONE AUTOMATICA DISABILITATA
   linea.stz[4].war[8..14] := FALSE;
   linea.stz[4].war[15] := FALSE;   // L1-ASPO[15]-M102 MADRINO -PRESENZA LAMIERA
   linea.stz[4].war[16..32] := FALSE;
   linea.stz[5].war[1..2] := FALSE;
   linea.stz[5].war[3] := FALSE;   // L1-RADDRIZZATRICE[3]-M141-FINE LAMIERA
   linea.stz[5].war[4..32] := FALSE;
   linea.stz[6].war[1..2] := FALSE;
   linea.stz[6].war[3] := FALSE;   // L1-GIUNZIONE[3]-CENTRALE OLEODINAMICA-MINIMO LIVELLO OLIO
   linea.stz[6].war[4..32] := FALSE;
   linea.stz[7].war[1..32] := FALSE;
   linea.stz[8].war[1..32] := FALSE;
   linea.stz[9].war[1..32] := FALSE;
   linea.stz[10].war[1..32] := FALSE;
   linea.stz[11].war[1..32] := FALSE;
   linea.stz[12].war[1..32] := FALSE;
   linea.stz[13].war[1..32] := FALSE;
   linea.stz[14].war[1..32] := FALSE;
   linea.stz[15].war[1..32] := FALSE;
   linea.stz[16].war[1..32] := FALSE;
   linea.stz[17].war[1..32] := FALSE;
   linea.stz[18].war[1..32] := FALSE;
   linea.stz[19].war[1..32] := FALSE;
   linea.stz[20].war[1..32] := FALSE;
   linea.stz[1..3].warningpc := 0;
   linea.stz[4].warningpc := 32;
   linea.stz[5..20].warningpc := 0;
END_DATA_BLOCK
